{attribute 'qualified_only'}
TYPE SEQUENCE_STEP :
(
	STEP_ERROR := -3,
	NO_STEP_CHANGE := -2,
	NO_STEP := -1,
	IDLE_STEP := 0,
	START_STEP := 1
);
END_TYPE
//  STEP_ERROR = '-3'
//  NO_STEP_CHANGE = '-2'
//  NO_STEP = '-1'

(* stored: Version 1.1.0.1
   EnumerationTextList SEQUENCE_STEP: Id {15fff023-6076-4274-bd71-f74277d76200} *)
